FUNCTION_BLOCK PUBLIC BeckHoff8xxxAxis_FB EXTENDS BeckHoffBasicAxis_FB  
VAR_INPUT		
	io_SafetyState: 	BYTE;	
END_VAR
VAR_IN_OUT	
END_VAR
VAR_OUTPUT	
END_VAR

VAR
//	DebugError					: UINT;
	Drive8000InitDone :BOOL := FALSE;
END_VAR

IF NOT Drive8000InitDone THEN
	Meth_Init();
	Drive8000InitDone := TRUE;
END_IF

AxisCtrlPtr^.Input.Parameter.Drive.eDriveType := enumDriveType.e8xxxBeckhoff;	
AxisCtrlPtr^.Input.Parameter.Drive.VendorNameID := eVendorNameID.Beckhoff;

SUPER^(AxisRef:=AxisRef);

AxisCtrlPtr^.Output.Status.DriveEnable:=	BYTE_TO_BOOL(io_SafetyState);

METHOD CreateDriveErrMsgDetails : enumMotorEvents
VAR_INPUT
	ErrorId			: UDINT;
END_VAR
CASE ErrorId OF
	
	16#0:
		CreateDriveErrMsgDetails := enumMotorEvents.NoEvents;
		fnLogMsg(ADR(LogMsg_0),LOG_ERROR,'Beckhoff Drive8 ErrorId %d  ,No error',UDINT_TO_DINT(ErrorId),0,0);
	16#2340: 
		CreateDriveErrMsgDetails := enumMotorEvents.MotorSupplyError ;
		fnLogMsg(ADR(LogMsg_0),LOG_ERROR,'Beckhoff Drive8 ErrorId %d  Short circuit (motor-side)',UDINT_TO_DINT(ErrorId),0,0);
	16#2380:
		CreateDriveErrMsgDetails := enumMotorEvents.MotorOverCurrent ;
		fnLogMsg(ADR(LogMsg_0),LOG_ERROR,'Beckhoff Drive8 ErrorId %d Continuous over current -U',UDINT_TO_DINT(ErrorId),0,0);
	16#2381:
		CreateDriveErrMsgDetails := enumMotorEvents.MotorOverCurrent ;
		fnLogMsg(ADR(LogMsg_0),LOG_ERROR,'Beckhoff Drive8 ErrorId %d Continuous over current - V',UDINT_TO_DINT(ErrorId),0,0);
	16#2382:
		CreateDriveErrMsgDetails := enumMotorEvents.MotorOverCurrent ;	
		fnLogMsg(ADR(LogMsg_0),LOG_ERROR,'Beckhoff Drive8 ErrorId %d Continuous over current Ohase W',UDINT_TO_DINT(ErrorId),0,0);
		
	16#2383:
		CreateDriveErrMsgDetails := enumMotorEvents.MotorSupplyError;
		fnLogMsg(ADR(LogMsg_0),LOG_ERROR,'Beckhoff Drive8 ErrorId %d Phase U current offset out of range',UDINT_TO_DINT(ErrorId),0,0);
	16#2384:
		CreateDriveErrMsgDetails := enumMotorEvents.MotorSupplyError;
		fnLogMsg(ADR(LogMsg_0),LOG_ERROR,'Beckhoff Drive8 ErrorId %d  Phase V current offset out of range',UDINT_TO_DINT(ErrorId),0,0);
	16#2385:
		CreateDriveErrMsgDetails := enumMotorEvents.MotorSupplyError;
		fnLogMsg(ADR(LogMsg_0),LOG_ERROR,'Beckhoff Drive8 ErrorId %d  Phase W current offset out of range',UDINT_TO_DINT(ErrorId),0,0);
	16#3180..16#3181 :
		CreateDriveErrMsgDetails := enumMotorEvents.MotorGeneralError;
		fnLogMsg(ADR(LogMsg_0),LOG_ERROR,'Beckhoff Drive8 ErrorId %d  Phase failure motor',UDINT_TO_DINT(ErrorId),0,0);
	16#3210: 
		CreateDriveErrMsgDetails := enumMotorEvents.MotorSupplyError;
		fnLogMsg(ADR(LogMsg_0),LOG_ERROR,'Beckhoff Drive ErrorId %d DC link overvoltage',UDINT_TO_DINT(ErrorId),0,0);
		
		
	16#3220:
		CreateDriveErrMsgDetails := enumMotorEvents.MotorSupplyError;
		fnLogMsg(ADR(LogMsg_0),LOG_ERROR,'Beckhoff Drive8 ErrorId %d DC-Link undervoltage',UDINT_TO_DINT(ErrorId),0,0);
	16#3280:
 		CreateDriveErrMsgDetails := enumMotorEvents.MotorSupplyError;
		fnLogMsg(ADR(LogMsg_0),LOG_ERROR,'Beckhoff Drive8 ErrorId %d 2  DC link is not ready',UDINT_TO_DINT(ErrorId),0,0);
	16#4310: 
		CreateDriveErrMsgDetails := enumMotorEvents.MotorOverTemp;
		fnLogMsg(ADR(LogMsg_0),LOG_ERROR,'Beckhoff Drive8 ErrorId %d Drive overtemperature ',UDINT_TO_DINT(ErrorId),0,0);
	16#4380:
		CreateDriveErrMsgDetails := enumMotorEvents.MotorOverTemp;
		fnLogMsg(ADR(LogMsg_0),LOG_ERROR,'Beckhoff Drive8 ErrorId %d  Fan speed seems to be zero',UDINT_TO_DINT(ErrorId),0,0);
	16#5112:
		CreateDriveErrMsgDetails := enumMotorEvents.MotorSupplyError;
		fnLogMsg(ADR(LogMsg_0),LOG_ERROR,'Beckhoff Drive8 ErrorId %d  Supply undervoltage: supply +24V',UDINT_TO_DINT(ErrorId),0,0);
		
	16#5180:
		CreateDriveErrMsgDetails := enumMotorEvents.DriveNotEnabled;
		fnLogMsg(ADR(LogMsg_0),LOG_ERROR,'Beckhoff Drive8 ErrorId %d Output stage STO active',UDINT_TO_DINT(ErrorId),0,0);
	16#5181:
		CreateDriveErrMsgDetails := enumMotorEvents.MotorSupplyError;
		fnLogMsg(ADR(LogMsg_0),LOG_ERROR,'Beckhoff Drive8 ErrorId %d Power supply controlword, torque off order',UDINT_TO_DINT(ErrorId),0,0);

	16#5182:
		CreateDriveErrMsgDetails := enumMotorEvents.MotorSupplyError;
		fnLogMsg(ADR(LogMsg_0),LOG_ERROR,'Beckhoff Drive8 ErrorId %d Power supply controlword, live counter inactive',UDINT_TO_DINT(ErrorId),0,0);

	16#5183:
		CreateDriveErrMsgDetails := enumMotorEvents.MotorSupplyError;
		fnLogMsg(ADR(LogMsg_0),LOG_ERROR,'Beckhoff Drive8 ErrorId %d Power supply controlword, NC handling order',UDINT_TO_DINT(ErrorId),0,0);
		
	16#5184:
		CreateDriveErrMsgDetails := enumMotorEvents.MotorSupplyError;
		fnLogMsg(ADR(LogMsg_0),LOG_ERROR,'Beckhoff Drive8 ErrorId %d  Supply DC link circuit is not ready',UDINT_TO_DINT(ErrorId),0,0);
	
	16#5185:
		CreateDriveErrMsgDetails := enumMotorEvents.MotorSupplyError;
		fnLogMsg(ADR(LogMsg_0),LOG_ERROR,'Beckhoff Drive8 ErrorId %d Power supply controlword, non-regenerative brake order',UDINT_TO_DINT(ErrorId),0,0);
	16#5186:
		CreateDriveErrMsgDetails := enumMotorEvents.MotorSupplyError;
		fnLogMsg(ADR(LogMsg_0),LOG_ERROR,'Beckhoff Drive8 ErrorId %d Power supply controlword, regenerative brake order',UDINT_TO_DINT(ErrorId),0,0);
		
	16#5187:
		CreateDriveErrMsgDetails := enumMotorEvents.MotorSupplyError;
		fnLogMsg(ADR(LogMsg_0),LOG_ERROR,'Beckhoff Drive8 ErrorId %d  Power supply communication is not established',UDINT_TO_DINT(ErrorId),0,0);
	16#5190:
		CreateDriveErrMsgDetails := enumMotorEvents.MotorSupplyError;
		fnLogMsg(ADR(LogMsg_0),LOG_ERROR,'Beckhoff Drive8 ErrorId %d  Test 5V supply failed',UDINT_TO_DINT(ErrorId),0,0);

	16#5192:
		CreateDriveErrMsgDetails := enumMotorEvents.MotorSupplyError;
		fnLogMsg(ADR(LogMsg_0),LOG_ERROR,'Beckhoff Drive8 ErrorId %d Supply overvoltage: supply +24V',UDINT_TO_DINT(ErrorId),0,0);

	
	16#5441:
		CreateDriveErrMsgDetails := enumMotorEvents.MotorPositionError;
		fnLogMsg(ADR(LogMsg_0),LOG_ERROR,'Beckhoff Drive8 ErrorId %d  Positive limit switch active',UDINT_TO_DINT(ErrorId),0,0);
	16#5442:
		CreateDriveErrMsgDetails := enumMotorEvents.DriveComError ;
		fnLogMsg(ADR(LogMsg_0),LOG_ERROR,'Beckhoff Drive8 ErrorId %d  Negative limit switch active',UDINT_TO_DINT(ErrorId),0,0);

	16#5580..16#6181:
		CreateDriveErrMsgDetails := enumMotorEvents.MotorGeneralError  ;
		fnLogMsg(ADR(LogMsg_0),LOG_ERROR,'Beckhoff Drive8 ErrorId %d Beckhoff internal Error',UDINT_TO_DINT(ErrorId),0,0);
	16#6182..16#6190:
		CreateDriveErrMsgDetails := enumMotorEvents.MotorGeneralError;
		fnLogMsg(ADR(LogMsg_0),LOG_ERROR,'Beckhoff Drive8 ErrorId %d  Internal Watchdog Error',UDINT_TO_DINT(ErrorId),0,0);
	16#6391..16#639F:
		CreateDriveErrMsgDetails := enumMotorEvents.PLCIllegalParam;
		fnLogMsg(ADR(LogMsg_0),LOG_ERROR,'Beckhoff Drive8 ErrorId %d Operation mode incompatible to PDO',UDINT_TO_DINT(ErrorId),0,0);
	16#63A2..16#63A5:
		CreateDriveErrMsgDetails := enumMotorEvents.MotorFeedBackErr;
		fnLogMsg(ADR(LogMsg_0),LOG_ERROR,'Beckhoff Drive8 ErrorId %d  No position offset',UDINT_TO_DINT(ErrorId),0,0);

	16#63A6..16#63B3:
		CreateDriveErrMsgDetails := enumMotorEvents.PLCIllegalParam ;
		fnLogMsg(ADR(LogMsg_0),LOG_ERROR,'Beckhoff Drive8 ErrorId %d  Jerk factor illegal',UDINT_TO_DINT(ErrorId),0,0);
	
	16#7180:
		CreateDriveErrMsgDetails := enumMotorEvents.MotorSupplyError ;
		fnLogMsg(ADR(LogMsg_0),LOG_ERROR,'Beckhoff Drive8 ErrorId %d Current monitoring error',UDINT_TO_DINT(ErrorId),0,0);


	16#7380:
		CreateDriveErrMsgDetails := enumMotorEvents.MotorSupplyError ;
		fnLogMsg(ADR(LogMsg_0),LOG_ERROR,'Beckhoff Drive8 ErrorId %d Current sensor motor phase U',UDINT_TO_DINT(ErrorId),0,0);
	16#7381:
		CreateDriveErrMsgDetails := enumMotorEvents.MotorSupplyError ;
		fnLogMsg(ADR(LogMsg_0),LOG_ERROR,'Beckhoff Drive8 ErrorId %d  Current sensor motor phase V',UDINT_TO_DINT(ErrorId),0,0);
	16#7382:
		CreateDriveErrMsgDetails := enumMotorEvents.MotorSupplyError ;
		fnLogMsg(ADR(LogMsg_0),LOG_ERROR,'Beckhoff Drive8 ErrorId %d  Current sensor motor phase W',UDINT_TO_DINT(ErrorId),0,0);
	16#8180:
		CreateDriveErrMsgDetails := enumMotorEvents.DriveComError ;
		fnLogMsg(ADR(LogMsg_0),LOG_ERROR,'Beckhoff Drive8 ErrorId %d System restart or sync lost',UDINT_TO_DINT(ErrorId),0,0);
	16#8181:	
		CreateDriveErrMsgDetails := enumMotorEvents.DriveComError ;
		fnLogMsg(ADR(LogMsg_0),LOG_ERROR,'Beckhoff Drive8 ErrorId %d Lost Distributed clocks Sync',UDINT_TO_DINT(ErrorId),0,0);

	16#8185:
		CreateDriveErrMsgDetails := enumMotorEvents.MotorGeneralError ;
		fnLogMsg(ADR(LogMsg_0),LOG_ERROR,'Beckhoff Drive8 ErrorId %d  need an extended fault reset command',UDINT_TO_DINT(ErrorId),0,0);
	16#8611:	
		CreateDriveErrMsgDetails := enumMotorEvents.MotorPositionError ;
		fnLogMsg(ADR(LogMsg_0),LOG_ERROR,'Beckhoff Drive8 ErrorId %d Following error',UDINT_TO_DINT(ErrorId),0,0);

	
	16#8A80..16#8A81:
		CreateDriveErrMsgDetails := enumMotorEvents.PLCIllegalParam ;
		fnLogMsg(ADR(LogMsg_0),LOG_ERROR,'Beckhoff Drive8 ErrorId %d  Illegal Modes Of Operation',UDINT_TO_DINT(ErrorId),0,0);
		
	16#A000..16#A00F :
		CreateDriveErrMsgDetails := enumMotorEvents.MotorGeneralError ;
		fnLogMsg(ADR(LogMsg_0),LOG_ERROR,'Beckhoff Drive8 ErrorId %d  Sync Manager Address Error',UDINT_TO_DINT(ErrorId),0,0);
	
	16#A010..16#A043 :
		CreateDriveErrMsgDetails := enumMotorEvents.PLCIllegalParam ;
		fnLogMsg(ADR(LogMsg_0),LOG_ERROR,'Beckhoff Drive8 ErrorId %d PDO/SDO Error',UDINT_TO_DINT(ErrorId),0,0);
	16#A082:
		CreateDriveErrMsgDetails := enumMotorEvents.MotorGeneralError ;
		fnLogMsg(ADR(LogMsg_0),LOG_ERROR,'Beckhoff Drive8 ErrorId %d  , EtherCAT Slave Stack Error',UDINT_TO_DINT(ErrorId),0,0);
	
	
	16#FF08:
		CreateDriveErrMsgDetails := enumMotorEvents.BreakResistorError ;
		fnLogMsg(ADR(LogMsg_0),LOG_ERROR,'Beckhoff Drive8 ErrorId %d  Shorted Coils Brake',UDINT_TO_DINT(ErrorId),0,0);
	16#FF0C:
		CreateDriveErrMsgDetails := enumMotorEvents.MotorGeneralError ;
		fnLogMsg(ADR(LogMsg_0),LOG_ERROR,'Beckhoff Drive8 ErrorId %d  TorqueOff with emergency brake',UDINT_TO_DINT(ErrorId),0,0);

	16#FFFF:
		CreateDriveErrMsgDetails := enumMotorEvents.MotorGeneralError;
		fnLogMsg(ADR(LogMsg_0),LOG_ERROR,'Beckhoff Drive8 ErrorId %d  Internal Error',UDINT_TO_DINT(ErrorId),0,0);
		
 	ELSE
		fnLogMsg(ADR(LogMsg_0),LOG_ERROR,'unknown Beckhoff Drive8 ErrorId %d ',UDINT_TO_DINT(ErrorId),0,0);
		CreateDriveErrMsgDetails := enumMotorEvents.NoEvents;
END_CASE
END_METHOD

METHOD GetErrCanAdrTemp : BOOL
VAR_INPUT
END_VAR
//Maybe this FB should be remove
CoeErrIdIndex		:= 16#583f;

		
//CoeErrIdIndex	:= 16#603F;
END_METHOD

METHOD Meth_Init : BOOL
VAR_INPUT
END_VAR
ErrorMSgSize := 64;
END_METHOD

END_FUNCTION_BLOCK

(* stored: Version 1.1.0.1, ProductVersion 3.1.4024.3
   POU BeckHoff8xxxAxis_FB: Id {2cb267e6-48a9-4a04-800a-fe261429fe20}, SpecialFunc None
   Method CreateDriveErrMsgDetails: Id {a94f66c2-fe74-446d-b8e5-cf524e217748}
   Method GetErrCanAdrTemp: Id {ad08e1f8-5c77-4da4-9b7d-9a6e1549dd25}
   Method Meth_Init: Id {fd716804-ac76-4b80-8a40-0cd70dbe5dda} *)
